# EPICS autosave request: iocBoot/iocE1608/auto_settings.req
file "E1608_settings.req", P=$(P)
